TYPE ST_InfoDataConnection :
STRUCT
	usiMapState	:USINT;
	usiMapDiag	:USINT;
	bySignal	:BYTE;
END_STRUCT
END_TYPE

(* stored: Version 1.1.0.1, ProductVersion 3.1.4024.12
   DUT ST_InfoDataConnection: Id {1852d4df-fee4-4d6a-8603-2a7502a29b2f} *)
